// TIA Portal V20 export
// export: Created 2026-07-10T11:12:35.9961376Z, ExportSetting WithDefaults, DisplayName Totally Integrated Automation Portal, DisplayVersion V20, DisplayName TIA Portal Openness, DisplayVersion V20, DisplayName TIA Portal Version Control Interface, DisplayVersion V20, DisplayName STEP 7 Professional, DisplayVersion V20, DisplayName STEP 7 Safety, DisplayVersion V20, DisplayName WinCC Basic/Comfort/Advanced, DisplayVersion V20, DisplayName WinCC Unified, DisplayVersion V20
VAR_GLOBAL   // PLC tag table "Default tag table"
   Doser1 AT %I0.0 : Bool;
   AlarmOpen1 AT %I0.1 : Bool;
   Doser2 AT %I0.2 : Bool;
   AlarmOpen2 AT %I0.3 : Bool;
   RunClose1 AT %I0.4 : Bool;
   RunOpen1 AT %I0.5 : Bool;
   RunClose2 AT %I0.6 : Bool;
   RunOpen2 AT %I0.7 : Bool;
   WaterCounterInPulse AT %I1.0 : Bool;
   WaterCounterOutPulse AT %I1.1 : Bool;
   AI0V AT %IW64 : Int;
   AI1V AT %IW66 : Int;
   AI0AV AT %IW128 : Int;
   AI1AV AT %IW130 : Int;
   AI2AV AT %IW132 : Int;
   AI3AV AT %IW134 : Int;
   AI4AV AT %IW80 : Int;
   PowerSupply AT %I1.2 : Bool;
   FlowAO AT %QW64 : Int;
   OutOpen1 AT %Q0.0 : Bool;
   OutClose1 AT %Q0.1 : Bool;
   OutOpen2 AT %Q0.2 : Bool;
   OutClose2 AT %Q0.3 : Bool;
   SirenOut AT %Q0.4 : Bool;
   System_Byte AT %MB1 : Byte;
   FirstScan AT %M1.0 : Bool;
   DiagStatusUpdate AT %M1.1 : Bool;
   AlwaysTRUE AT %M1.2 : Bool;
   AlwaysFALSE AT %M1.3 : Bool;
   Clock_Byte AT %MB0 : Byte;
   Clock_10Hz AT %M0.0 : Bool;
   Clock_5Hz AT %M0.1 : Bool;
   "Clock_2.5Hz" AT %M0.2 : Bool;
   Clock_2Hz AT %M0.3 : Bool;
   "Clock_1.25Hz" AT %M0.4 : Bool;
   Clock_1Hz AT %M0.5 : Bool;
   "Clock_0.625Hz" AT %M0.6 : Bool;
   "Clock_0.5Hz" AT %M0.7 : Bool;
   Damper1_AutoMode AT %I1.3 : Bool;
   Damper2_AutoMode AT %I1.4 : Bool;
   OsmosOut AT %Q0.5 : Bool;
   OsmosAO AT %QW66 : Int;
   DoserOut AT %Q0.6 : Bool;
   ChlorationOut AT %Q0.7 : Bool;
END_VAR
